{attribute 'enable_dynamic_creation'}
// Provides array helper methods for easier work with arrays accross programming.
PROGRAM ArrayHelper

// Clears the entire array. Returns TRUE if operation was sucessfull.
METHOD PUBLIC Clear : BOOL
VAR_INPUT
	arr			: ANY;	// Array to be cleared
END_VAR
IF NOT ValidateArrayVar(arr) THEN
	RETURN;
END_IF

Tc2_System.MEMSET(
	destAddr := arr.pValue,
	fillByte := 0,
	n := DINT_TO_UDINT(arr.diSize));
	
Clear := TRUE;
END_METHOD

// Looks trough the array and returns TRUE if any element equals to the one provided.
METHOD DoesArrayContainItem : BOOL
VAR_INPUT
	arr		: ANY;	// Array to be checked
	item	: ANY;	// Item to be found in the array
END_VAR

VAR
	itemCount	: T_ArrayIndexer;
	currentItem	: T_ArrayIndexer;
	cmpResult	: E_MemCmpResults;
END_VAR
IF NOT ValidateArrayVar(arr) THEN
	RETURN;
END_IF

IF item.diSize = 0 OR_ELSE	// If item size is 0
	(arr.diSize MOD item.diSize) <> 0 	// If incorrect item is provided (division will return non 0 remainder)
THEN
	RETURN;
END_IF

itemCount := arr.diSize/item.diSize;

FOR currentItem := 0 TO itemCount - 1 BY 1 DO
	cmpResult := Tc2_System.MEMCMP(
		pBuf1 := arr.pValue + DINT_TO_DWORD(currentItem * item.diSize),
		pBuf2 := item.pValue,
		n := DINT_TO_UDINT(item.diSize));
		
	IF cmpResult = E_MemCmpResults.IDENTICAL THEN
		DoesArrayContainItem := TRUE;
		RETURN;
	END_IF
END_FOR
END_METHOD

// Looks trough the array and return the last non-zero element to the result variable.
// Returns TRUE if an element was found and FALSE if no empty elements are found.
// Note that this method uses memmory allocation. All occupied memory is released after method finishes.
METHOD PUBLIC FindLastOccupiedItem	: BOOL
VAR_INPUT
	arr			: ANY;	// Array to look for the last element value
	dataType	: ANY;	// Data type of the array elements, can be used like this : datayType := arr[0]
	result		: ANY;	// Result variable, result be written to this variable
END_VAR

VAR
	i								: T_ArrayIndexer;
	maxIndex						: T_ArrayIndexer;
	compareResult					: E_MemCmpResults;
	ptrAllocatedBytes_emptyElement	: POINTER TO BYTE;
END_VAR
IF NOT ValidateArrayVar(arr) OR result.TypeClass <> dataType.TypeClass THEN
	RETURN;
END_IF

maxIndex :=  GetElementCount(arr := arr, dataType := dataType) - 1;
ptrAllocatedBytes_emptyElement := __NEW(BYTE, DINT_TO_UDINT(dataType.diSize));

// Array with 1 element - loop would point to invalid position, exit early by just checking the values
IF maxIndex = 0 THEN
	IF arr.pValue^ <> ptrAllocatedBytes_emptyElement^ THEN
		Tc2_System.MEMCPY(
			srcAddr := arr.pValue,
			destAddr := result.pValue,
			n := DINT_TO_UDINT(dataType.diSize));
			FindLastOccupiedItem := TRUE;
	END_IF
	// Delete allocated memory and return from the method
	__DELETE(ptrAllocatedBytes_emptyElement);
	RETURN;
END_IF

FOR i := maxIndex TO 0 BY -1 DO
	compareResult := Tc2_System.MEMCMP(
		pBuf1 := arr.pValue +  DINT_TO_DWORD(i * dataType.diSize),
		pBuf2 := ptrAllocatedBytes_emptyElement,
		n := DINT_TO_UDINT(dataType.diSize));
		
	// If element is not empty, return
	IF compareResult <> E_MemCmpResults.IDENTICAL THEN
		Tc2_System.MEMCPY(
			srcAddr := arr.pValue +  DINT_TO_DWORD(i * dataType.diSize),
			destAddr := result.pValue,
			n := DINT_TO_UDINT(dataType.diSize));
		FindLastOccupiedItem := TRUE;
		EXIT;
	END_IF
END_FOR

// Delete allocated memory
__DELETE(ptrAllocatedBytes_emptyElement);
END_METHOD

// Returns the number of elements in the array.
METHOD PUBLIC GetElementCount : DINT
VAR_INPUT
	arr			: ANY;	// Array to be checked.
	dataType	: ANY;	// Data type of the array elements, can be used like this : datayType := arr[0]
END_VAR
IF ValidateArrayVar(arr) = FALSE THEN
	RETURN;
END_IF

IF dataType.diSize = 0 THEN
	RETURN;
END_IF
GetElementCount := arr.diSize / dataType.diSize;
END_METHOD

// Gets the maximum array index that can be used for looping or index accessing
METHOD PUBLIC GetMaxIndex : DINT
VAR_INPUT
	arr			: ANY;	// Array to be checked.
	dataType	: ANY;	// Data type of the array elements, can be used like this : datayType := arr[0]
	startIndex	: T_ArrayIndexer;
END_VAR
IF ValidateArrayVar(arr) = FALSE THEN
	RETURN;
END_IF

GetMaxIndex := startIndex + GetElementCount(arr := arr, dataType := dataType) - 1;
END_METHOD

// Inserts the item to the start of the array. 
// Array contents are shifted by 1, last item is deleted.
METHOD InsertAtStart : BOOL
VAR_INPUT	
	arr		: ANY;	// Array to be checked.
	item	: ANY;	// Item to be inserted on start
 END_VAR
IF ValidateArrayVar(arr) = FALSE THEN
	RETURN;
END_IF

ShiftUp(
	arr := arr,
	dataType := item);

// Set first element value
Tc2_System.MEMCPY(
	destAddr := arr.pValue,
	srcAddr := item.pValue,
	n := DINT_TO_UDINT(item.diSize));
END_METHOD

// Iterates the array and sets the value when first empty slot is found. 
// Note that this method uses memmory allocation. All occupied memory is released after method finishes.
METHOD SetAtFirstEmptySlot
VAR_INPUT
	arr		: ANY;	// Array to be checked.
	item	: ANY;	// Item to set
END_VAR

VAR
	ptrByte 			: POINTER TO BYTE;
	i					: T_ArrayIndexer;
	maxIndex			: T_ArrayIndexer;
	ptrAllocatedBytes	: POINTER TO BYTE;
	cmpResult			: DINT;
END_VAR
IF ValidateArrayVar(arr) = FALSE THEN
	RETURN;
END_IF

maxIndex :=  GetElementCount(arr := arr, dataType := item) - 1;
ptrAllocatedBytes := __NEW(BYTE, DINT_TO_UDINT(arr.diSize));

FOR i := 0 TO maxIndex BY 1 DO
	ptrByte := arr.pValue + DINT_TO_UDINT(item.diSize * i);	
	
	cmpResult := Tc2_System.MEMCMP(
			n := DINT_TO_UDINT(item.diSize),
			pBuf1 := ptrAllocatedBytes,
			pBuf2 := ptrByte);
			
	IF cmpResult = E_MemCmpResults.IDENTICAL THEN
		Tc2_System.MEMCPY(
			destAddr := ptrByte,
			n := DINT_TO_UDINT(item.diSize),
			srcAddr := item.pValue);
		EXIT;
	END_IF
END_FOR

__DELETE(ptrAllocatedBytes);
END_METHOD

// Shifts the array down, losing first element and clearing last element in the process.
METHOD ShiftDown
VAR_INPUT
	arr		: ANY;	// Array to be checked.
	dataType	: ANY;	// Data type of the array elements, can be used like this : datayType := arr[0]
END_VAR
IF ValidateArrayVar(arr) = FALSE THEN
	RETURN;
END_IF

Tc2_System.MEMMOVE(	
	destAddr := arr.pValue,
	srcAddr := arr.pValue + DINT_TO_UDINT(dataType.diSize),
	n := DINT_TO_UDINT(arr.diSize - dataType.diSize));

// Clear last element
Tc2_System.MEMSET(
	fillByte := 0,
	n := DINT_TO_UDINT(dataType.diSize),
	destAddr := arr.pValue + DINT_TO_UDINT(arr.diSize - dataType.diSize));
END_METHOD

// Shifts the array up, losing last element and clearing first element in the process.
METHOD ShiftUp
VAR_INPUT
	arr			: ANY;	// Array to be checked.
	dataType	: ANY;	// Data type of the array elements, can be used like this : datayType := arr[0]
END_VAR
IF ValidateArrayVar(arr) = FALSE THEN
	RETURN;
END_IF


Tc2_System.MEMMOVE(
	destAddr := arr.pValue + DINT_TO_UDINT(dataType.diSize),
	srcAddr := arr.pValue,
	n := DINT_TO_UDINT(arr.diSize - dataType.diSize));

// Clear first element
Tc2_System.MEMSET(
	fillByte := 0,
	n := DINT_TO_UDINT(dataType.diSize),
	destAddr := arr.pValue);
END_METHOD

METHOD PRIVATE ValidateArrayVar : BOOL
VAR_INPUT
	arr	: ANY;
END_VAR
VAR
	isArray		: BOOL;
	isReference	: BOOL;
END_VAR
isArray := F_DoesVarTypeEqual(arr, IBaseLibrary.TYPE_ARRAY);
isReference := F_DoesVarTypeEqual(arr, IBaseLibrary.TYPE_REFERENCE);

ValidateArrayVar := isArray OR isReference;
END_METHOD

END_PROGRAM

(* stored: Version 1.1.0.1, ProductVersion 3.1.4024.15
   POU ArrayHelper: Id {1d7a0d08-3c88-00ea-2870-5cdbd9795f9a}, SpecialFunc None
   Method Clear: Id {be15889c-c0e1-09a6-20bb-cafe31f0b982}
   Method DoesArrayContainItem: Id {4bfa90e6-378d-00b9-19dc-21db7c691e2f}
   Method FindLastOccupiedItem: Id {e804b769-2043-0cee-39f9-86bb16a4f8d7}
   Method GetElementCount: Id {be71fb45-3c58-0314-18ef-9118e35efd5e}
   Method GetMaxIndex: Id {edabc55d-cc53-030c-3bc1-e981a29138e7}
   Method InsertAtStart: Id {0f3f90b7-bf52-0373-102d-0814471c7b79}
   Method SetAtFirstEmptySlot: Id {8d93fb02-0d20-05a7-18f0-70a436d31e09}
   Method ShiftDown: Id {bf9c2e03-6302-0e64-05d0-eb3dbb49d451}
   Method ShiftUp: Id {55cff527-a1ec-0ba7-3953-cd8958d2ceb2}
   Method ValidateArrayVar: Id {b9ef476c-b27f-0470-04c9-84ac8b60f534} *)
